INTERFACE I_ModeProvider

// 0 = Idle, 1 = Auto, 2 = Manual, 3 = Paused (added at CR-1)
PROPERTY CurrentMode : INT
GET
END_GET
END_PROPERTY

PROPERTY AllowRun : BOOL
GET
END_GET
END_PROPERTY

PROPERTY AllowJog : BOOL
GET
END_GET
END_PROPERTY

END_INTERFACE

(* stored: Version 1.1.0.1
   Itf I_ModeProvider: Id {2dc23b51-a2b2-47d1-a42e-5650f2ad2c8a}
   Property CurrentMode: Id {0adc6758-8186-4c90-be8e-35cede23ba37}
   Get Get: Id {00a75fab-d1eb-41b6-b9e8-cba987909e02}
   Property AllowRun: Id {39711bd7-01fe-4cf9-b463-33b2b0d6cb0a}
   Get Get: Id {801baaa9-fff2-42f4-bcbf-1770412db082}
   Property AllowJog: Id {1d3aa30d-9b91-492d-b641-15ee60c38099}
   Get Get: Id {c932edbc-30b0-4102-b904-28af96c097ad} *)
